ORGANIZATION_BLOCK MAIN:OB1
TITLE=中文详细注释版
// 文件说明：本文件只完善中文注释，不改变 PLC 指令、地址和执行顺序。
// 编码说明：本文件采用 GBK/ANSI 编码，供现场 PLC 编辑环境直接打开。
//
// ======================== 本项目工序与地址总表 ========================
// 说明：“程序网络 N”是 AWL Network 编号，不等于设备主屏上的工序序号。
// 主工序顺序（与上位机主屏一致）：
//   等待启动(M0.0=0) -> 初始位垂直复位(M10.0) -> 初始位确认(M10.1)
//   -> 检测区1定位(M10.2) -> 热源位夹具下压(M10.3) -> 30秒稳定 -> 30秒噪声采集(M25.2)
//   -> 热源干扰测试(M10.4)
//   -> 热源后夹具上升(M10.5) -> 检测区2定位(M10.6) -> 爆闪位夹具下压(M10.7)
//   -> 五次爆闪测试(M11.0) -> 电磁干扰(M11.2) -> 回初始位确认(M11.4)
//   -> 流程完成(M0.1)。
//
// 输入 I（现场反馈/命令）：
//   I0.0 初始位置传感器；I0.2 检测区1位置传感器；I0.1 检测区2位置传感器。
//   I0.4 垂直下限反馈；I0.3 垂直上限反馈（本版主链以定时到位为主，地址保留作项目对照）。
//   I1.0 安全/急停输入：1=安全链满足，0=急停或安全链断开。
//   I1.3 自动启动输入：闭合上升沿触发一次完整检测工序。
//
// 物理输出继电器 Q（与主屏“输出继电器 Q”一致）：
//   Q0.0 预留/本程序无独立驱动，仅在总复位时清零。
//   Q0.1 模拟人温度/热源；Q0.2、Q0.3 预留/本程序无独立驱动。
//   Q0.4 上下电机总电源；Q0.5 左右电机运行；Q0.6 左右电机停止。
//   Q0.7 电磁干扰继电器，实际链路为 M11.2 AND M31.7 -> Q0.7。
//   Q1.0 气缸/挥手测试；Q1.1 垂直方向（1=上，0=下）。
//   Q1.2 爆闪灯1；Q1.3 爆闪灯2。
//
// 主状态与启动/停止辅助继电器 M：
//   M0.0 自动运行；M0.1 流程完成；M0.2 流程报警；M0.3 安全链满足。
//   M1.0 停止/中止锁存；M1.2 启动条件确认后的单扫描启动脉冲。
//   M1.5 启动请求上一扫描状态；M1.6 启动请求上升沿；M1.7 手动使能启动通道。
//   M2.0 停止请求；M2.1 总复位/初始化请求；M2.2 安全限位；
//   M2.3 启动请求；M2.4 手动使能。M20.0 为安全链断开故障镜像。
//
// 主工序步进继电器（同一时刻通常只保持当前工序位）：
//   M10.0 初始位垂直复位；M10.1 初始位确认；M10.2 检测区1定位。
//   M10.3 热源位夹具下压；M10.4 热源干扰测试；M10.5 热源后夹具上升。
//   M10.6 检测区2定位；M10.7 爆闪位夹具下压；M11.0 五次爆闪测试。
//   M11.1 外部/备用的电磁工序启动脉冲；M11.2 电磁干扰工序控制位；
//   M11.3 回零完成后的流程结束脉冲；M11.4 电磁干扰后回初始位标志。
//
// 工序完成条件与动作子步：
//   M12.0 初始垂直复位延时完成；M12.1 初始位置确认；M12.2 检测区1到位。
//   M12.3 热源位夹具下压延时完成；M12.5 热源后夹具上升延时完成；
//   M12.6 检测区2到位；M12.7 爆闪位夹具下压延时完成。
//   M13.0~M13.4 热源干扰时的气缸/挥手脉冲子步（开、关交替）。
//   M13.5~M15.7 五次爆闪时序子步；奇数发光段驱动 Q1.2、Q1.3，间隔段熄灯。
//   M14.0 初始复位后的重叠移动等待；M14.1 初始位至检测区1的启动等待；
//   M14.2 检测区1到位后的下压启动等待；M14.3 上升后的水平移动等待（预留链）；
//   M14.4 检测区2到位后的下压启动等待。
//   M15.0 热源位下压后的稳定等待标志；M15.1 爆闪位下压后的稳定等待标志；
//   M15.2 热源测试后“垂直上升+水平移向检测区2”的重叠动作标志；
//   M15.3 热源夹具上升完成、等待进入检测区2下压的衔接标志。
//
// 上位机/通讯状态与事件留痕位：
//   M21.0 初始位阶段；M21.1 检测区1/热源阶段；M21.2 检测区2/爆闪阶段；
//   M21.3 电磁干扰阶段；M21.4 初始位置已确认；M21.5 热源后夹具已上升；
//   M21.6 五次爆闪已完成；M21.7 电磁干扰已完成。
//   M22.0 初始垂直复位完成；M22.1、M22.2 初始位置确认留痕；
//   M22.3 检测区1到位；M22.4 热源位下压完成；M22.5 热源干扰完成；
//   M22.6 爆闪位下压完成；M22.7 运动到位/衔接留痕（由上升或检测区2到位置位）。
//   M23.0 五次爆闪完成；M23.1 电磁干扰开始；M23.2 电磁干扰完成；
//   M23.3 电磁干扰完成后开始回初始位。
//
// 自动/手动动作命令、沿检测及安全合成：
//   M29.0 自动左右运行；M29.1 自动垂直下行；M29.2 自动垂直上行；
//   M29.3 自动气缸/挥手；M29.4 自动爆闪命令（当前五次爆闪另由时序子步直接合成）。
//   M30.0~M30.6 手动/调试动作命令；M30.7 手动总停止/全部输出清零。
//   M28.0~M28.4 保存 M29.0~M29.4 的上一扫描状态；
//   M26.0~M26.4 为相应自动动作的上升沿，M27.0~M27.4 为下降沿；
//   M26.5 为任一自动动作上升沿，M27.5 为垂直上/下动作结束的互锁辅助位。
//   M31.0 热源输出合成；M31.1 垂直电源合成；M31.2 垂直向上方向合成；
//   M31.3 水平运行合成；M31.4 水平停止合成；M31.5 爆闪灯1合成；
//   M31.6 爆闪灯2合成；M31.7 总输出安全使能（安全链满足且无手动总停止）。
//   M25.0 安全限位上升沿单扫描脉冲；M25.1 正常水平停止请求；
//   M25.2 为信号稳定后的30秒噪声采集窗口，由 T63 稳定到时后直接驱动。
//
// 状态字：VW600=上位机工序阶段码；VW602=上位机工序子步码。
//
// ======================== 定时器实际时间参数表 ========================
// 计时规则：本程序全部使用 TON T37~T63；按 S7-200 SMART 定时器规则，
//           T37~T63 的时间基准均为 100 ms，实际延迟 = PT预置值 x 0.1秒。
//           下表按本文件当前 PT 值换算；修改 PT 后必须同步更新此表及网络注释。
//
// 初始位、定位及夹具动作：
//   T44  初始位垂直复位动作延时       PT=+20   -> 2.0秒
//   T45  热源位夹具下压动作延时       PT=+100  -> 10.0秒
//   T46  热源测试后夹具上升动作延时   PT=+100  -> 10.0秒
//   T47  爆闪位夹具下压动作延时       PT=+100  -> 10.0秒
//
// 工序切换及机械稳定等待：
//   T48  初始复位后的重叠移动等待     PT=+80   -> 8.0秒
//   T49  初始位至检测区1启动等待      PT=+10   -> 1.0秒
//   T50  检测区1到位后的下压启动等待  PT=+10   -> 1.0秒
//   T51  信号稳定后噪声采集窗口   PT=+300  -> 30.0秒
//   T52  检测区2到位后的下压切换等待  PT=+10   -> 1.0秒
//   T62  垂直上升与水平移动重叠许可   PT=+20   -> 2.0秒
//   T63  热源位夹具下压后的稳定等待 PT=+300  -> 30.0秒
//   T38  爆闪位夹具下压后的稳定等待 PT=+100  -> 10.0秒
//
// 热源干扰/气缸挥手节拍：
//   T37、T40、T41、T42、T43 每段 PT=+10 -> 每段1.0秒；
//   共5段、总时序约5.0秒，形成3次动作段与2次间隔段。
//
// 五次爆闪节拍：
//   T53~T61 共9段，每段 PT=+10 -> 每段1.0秒；
//   总时序约9.0秒，形成5次亮灯段与4次灭灯间隔段。
//
// 电磁干扰：
//   T39  电磁干扰继电器 Q0.7 保持时间 PT=+100 -> 10.0秒。
// ======================================================================
// ======================================================================
BEGIN
// ----------------------------------------------------------------------
// 安全链、报警及复位总控
// ----------------------------------------------------------------------
Network 1
// 程序网络 1：把安全/急停输入 I1.0 映射为“安全链满足”M0.3。
// 输入状态初始化。
// 装载 I1.0 的状态，作为当前逻辑判断起点。
LD     I1.0
// 将当前逻辑结果写入 M0.3。
=      M0.3
Network 2
// 程序网络 2：安全链断开或收到停止请求时，生成停止/中止锁存 M1.0。
// 装载 I1.0 的反状态，作为当前逻辑判断起点。
LDN    I1.0
// 与 M2.0 进行并联“或”条件判断。
O      M2.0
// 将当前逻辑结果写入 M1.0。
=      M1.0
Network 3
// 程序网络 3：将安全链断开状态镜像到故障辅助位 M20.0。
// 装载 I1.0 的反状态，作为当前逻辑判断起点。
LDN    I1.0
// 将当前逻辑结果写入 M20.0。
=      M20.0
Network 4
// 程序网络 4：安全链断开时置流程报警 M0.2。
// 装载 M20.0 的状态，作为当前逻辑判断起点。
LD     M20.0
// 将当前逻辑结果写入 M0.2。
=      M0.2
Network 5
// 程序网络 5：执行流程条件判断与状态控制。
// 装载 M2.1 的状态，作为当前逻辑判断起点。
LD     M2.1
// 条件成立时复位 M0.0，连续复位 3 位。
R      M0.0, 3
Network 6
// 程序网络 6：满足条件时执行批量复位/停止处理。
// 装载 M2.1 的状态，作为当前逻辑判断起点。
LD     M2.1
// 条件成立时复位 M10.0，连续复位 12 位。
R      M10.0, 12
// 条件成立时复位 M11.4，连续复位 1 位。
R      M11.4, 1
// 条件成立时复位 M13.0，连续复位 8 位。
R      M13.0, 8
// 条件成立时复位 M14.0，连续复位 8 位。
R      M14.0, 8
// 条件成立时复位 M15.0，连续复位 4 位。
R      M15.0, 4
// 条件成立时复位 M15.4，连续复位 4 位。
R      M15.4, 4
Network 7
// 程序网络 7：执行流程条件判断与状态控制。
// 装载 M2.1 的状态，作为当前逻辑判断起点。
LD     M2.1
// 条件成立时复位 M12.0，连续复位 10 位。
R      M12.0, 10
Network 8
// 程序网络 8：满足条件时执行批量复位/停止处理。
// 装载 M2.1 的状态，作为当前逻辑判断起点。
LD     M2.1
// 条件成立时复位 M21.0，连续复位 8 位。
R      M21.0, 8
// 条件成立时复位 M29.0，连续复位 8 位。
R      M29.0, 8
// 条件成立时复位 M30.0，连续复位 8 位。
R      M30.0, 8
// 条件成立时复位 Q0.0，连续复位 8 位。
R      Q0.0, 8
// 条件成立时复位 Q1.0，连续复位 4 位。
R      Q1.0, 4
Network 9
// 程序网络 9：执行流程条件判断与状态控制。
// 装载 M2.1 的状态，作为当前逻辑判断起点。
LD     M2.1
// 条件成立时复位 M22.0，连续复位 12 位。
R      M22.0, 12
Network 10
// 程序网络 10：执行流程条件判断与状态控制。
// 装载 M2.1 的状态，作为当前逻辑判断起点。
LD     M2.1
// 条件成立时复位 M20.0，连续复位 1 位。
R      M20.0, 1
Network 11
// 程序网络 11：更新流程状态字或显示/通讯状态值。
// 装载 M2.1 的状态，作为当前逻辑判断起点。
LD     M2.1
// 条件成立时将字数据 +0 写入 VW600。
MOVW   +0, VW600
Network 12
// 程序网络 12：更新流程状态字或显示/通讯状态值。
// 装载 M2.1 的状态，作为当前逻辑判断起点。
LD     M2.1
// 条件成立时将字数据 +0 写入 VW602。
MOVW   +0, VW602
Network 13
// 程序网络 13：执行流程条件判断与状态控制。
// 装载 M1.0 的状态，作为当前逻辑判断起点。
LD     M1.0
// 条件成立时复位 M0.0，连续复位 1 位。
R      M0.0, 1
Network 14
// 程序网络 14：满足条件时执行批量复位/停止处理。
// 装载 M1.0 的状态，作为当前逻辑判断起点。
LD     M1.0
// 条件成立时复位 M10.0，连续复位 12 位。
R      M10.0, 12
// 条件成立时复位 M11.4，连续复位 1 位。
R      M11.4, 1
// 条件成立时复位 M13.0，连续复位 8 位。
R      M13.0, 8
// 条件成立时复位 M14.0，连续复位 8 位。
R      M14.0, 8
// 条件成立时复位 M15.0，连续复位 4 位。
R      M15.0, 4
// 条件成立时复位 M15.4，连续复位 4 位。
R      M15.4, 4
Network 15
// 程序网络 15：执行流程条件判断与状态控制。
// 装载 M1.0 的状态，作为当前逻辑判断起点。
LD     M1.0
// 条件成立时复位 M12.0，连续复位 10 位。
R      M12.0, 10
Network 16
// 程序网络 16：满足条件时执行批量复位/停止处理。
// 装载 M1.0 的状态，作为当前逻辑判断起点。
LD     M1.0
// 条件成立时复位 M21.0，连续复位 8 位。
R      M21.0, 8
// 条件成立时复位 M22.0，连续复位 12 位。
R      M22.0, 12
// 条件成立时复位 M29.0，连续复位 8 位。
R      M29.0, 8
// 条件成立时复位 M30.0，连续复位 8 位。
R      M30.0, 8
// 条件成立时复位 Q0.0，连续复位 8 位。
R      Q0.0, 8
// 条件成立时复位 Q1.0，连续复位 4 位。
R      Q1.0, 4
Network 17
// 程序网络 17：更新流程状态字或显示/通讯状态值。
// 装载 M1.0 的状态，作为当前逻辑判断起点。
LD     M1.0
// 条件成立时将字数据 +0 写入 VW600。
MOVW   +0, VW600
Network 18
// 程序网络 18：更新流程状态字或显示/通讯状态值。
// 装载 M1.0 的状态，作为当前逻辑判断起点。
LD     M1.0
// 条件成立时将字数据 +0 写入 VW602。
MOVW   +0, VW602
// ----------------------------------------------------------------------
// 启动请求沿检测与自动流程起动
// ----------------------------------------------------------------------
Network 19
// 程序网络 19：组合条件并生成状态或输出结果。
// 装载 M2.3 的状态，作为当前逻辑判断起点。
LD     M2.3
// 与 M1.5 的反状态进行串联条件判断。
AN     M1.5
// 将当前逻辑结果写入 M1.6。
=      M1.6
Network 20
// 程序网络 20：组合条件并生成状态或输出结果。
// 装载 M2.3 的状态，作为当前逻辑判断起点。
LD     M2.3
// 将当前逻辑结果写入 M1.5。
=      M1.5
Network 21
// 程序网络 21：组合条件并生成状态或输出结果。
// 装载 M1.6 的状态，作为当前逻辑判断起点。
LD     M1.6
// 与 M2.4 进行串联条件判断。
A      M2.4
// 与 M0.3 进行串联条件判断。
A      M0.3
// 将当前逻辑结果写入 M1.7。
=      M1.7
Network 22
// 程序网络 22：合成自动/手动启动条件，输出一次启动确认脉冲 M1.2。
// I1.3 上升沿通过正常安全联锁后启动自动流程。
// 装载 M1.6 的状态，作为当前逻辑判断起点。
LD     M1.6
// 与 M0.3 进行串联条件判断。
A      M0.3
// 与 M0.2 的反状态进行串联条件判断。
AN     M0.2
// 与 M0.0 的反状态进行串联条件判断。
AN     M0.0
// 与 M1.7 进行并联“或”条件判断。
O      M1.7
// 装载 I1.3 的状态，作为当前逻辑判断起点。
LD     I1.3
// 检测当前逻辑结果的上升沿，仅在上升沿扫描周期成立。
EU
// 与 M0.3 进行串联条件判断。
A      M0.3
// 与 M0.2 的反状态进行串联条件判断。
AN     M0.2
// 与 M0.0 的反状态进行串联条件判断。
AN     M0.0
// 将当前逻辑块与前一逻辑块进行“或”运算。
OLD
// 将当前逻辑结果写入 M1.2。
=      M1.2
Network 23
// 程序网络 23：执行流程条件判断与状态控制。
// 装载 M1.2 的状态，作为当前逻辑判断起点。
LD     M1.2
// 条件成立时置位 M0.0，连续置位 1 位。
S      M0.0, 1
Network 24
// 程序网络 24：执行流程条件判断与状态控制。
// 装载 M1.2 的状态，作为当前逻辑判断起点。
LD     M1.2
// 条件成立时复位 M0.1，连续复位 1 位。
R      M0.1, 1
Network 25
// 程序网络 25：满足条件时执行批量复位/停止处理。
// 装载 M1.2 的状态，作为当前逻辑判断起点。
LD     M1.2
// 条件成立时复位 M10.0，连续复位 12 位。
R      M10.0, 12
// 条件成立时复位 M11.4，连续复位 1 位。
R      M11.4, 1
// 条件成立时复位 M13.0，连续复位 8 位。
R      M13.0, 8
// 条件成立时复位 M14.0，连续复位 8 位。
R      M14.0, 8
// 条件成立时复位 M15.0，连续复位 4 位。
R      M15.0, 4
// 条件成立时复位 M15.4，连续复位 4 位。
R      M15.4, 4
Network 26
// 程序网络 26：执行流程条件判断与状态控制。
// 装载 M1.2 的状态，作为当前逻辑判断起点。
LD     M1.2
// 条件成立时复位 M2.0，连续复位 1 位。
R      M2.0, 1
Network 27
// 程序网络 27：满足条件时执行批量复位/停止处理。
// 装载 M1.2 的状态，作为当前逻辑判断起点。
LD     M1.2
// 条件成立时复位 M21.0，连续复位 8 位。
R      M21.0, 8
// 条件成立时复位 M29.0，连续复位 8 位。
R      M29.0, 8
// 条件成立时复位 M30.0，连续复位 8 位。
R      M30.0, 8
// 条件成立时复位 Q0.0，连续复位 8 位。
R      Q0.0, 8
// 条件成立时复位 Q1.0，连续复位 4 位。
R      Q1.0, 4
Network 28
// 程序网络 28：执行流程条件判断与状态控制。
// 装载 M1.2 的状态，作为当前逻辑判断起点。
LD     M1.2
// 条件成立时复位 M22.0，连续复位 12 位。
R      M22.0, 12
Network 29
// 程序网络 29：启动后进入“初始位垂直复位”M10.0，并发出自动上行 M29.2。
// 装载 M1.2 的状态，作为当前逻辑判断起点。
LD     M1.2
// 条件成立时置位 M10.0，连续置位 1 位。
S      M10.0, 1
// 条件成立时置位 M29.2，连续置位 1 位。
S      M29.2, 1
Network 30
// 程序网络 30：更新流程状态字或显示/通讯状态值。
// 装载 M1.2 的状态，作为当前逻辑判断起点。
LD     M1.2
// 条件成立时将字数据 +1 写入 VW600。
MOVW   +1, VW600
Network 31
// 程序网络 31：更新流程状态字或显示/通讯状态值。
// 装载 M1.2 的状态，作为当前逻辑判断起点。
LD     M1.2
// 条件成立时将字数据 +1 写入 VW602。
MOVW   +1, VW602
// ----------------------------------------------------------------------
// 主工序完成条件、延时及到位判定
// ----------------------------------------------------------------------
Network 32
// 程序网络 32：执行流程条件判断与状态控制。
// 装载 M10.1 的状态，作为当前逻辑判断起点。
LD     M10.1
// 与 M10.2 进行并联“或”条件判断。
O      M10.2
// 与 M10.6 进行并联“或”条件判断。
O      M10.6
// 条件成立时复位 Q0.6，连续复位 1 位。
R      Q0.6, 1
// 条件成立时置位 M29.0，连续置位 1 位。
S      M29.0, 1
Network 33
// 程序网络 33：初始位垂直复位动作计时 T44。
// 垂直机构初始化：先执行上行定时，再与水平回零流程进行重叠动作。
// 装载 M10.0 的状态，作为当前逻辑判断起点。
LD     M10.0
// T44（初始位垂直复位动作延时）：PT=+20，时间基准=100 ms，实际延迟=2.0秒。
TON    T44, +20
Network 34
// 程序网络 34：T44 到时，生成初始垂直复位完成 M12.0。
// 装载 T44 的状态，作为当前逻辑判断起点。
LD     T44
// 将当前逻辑结果写入 M12.0。
=      M12.0
Network 35
// 程序网络 35：M10.1 期间检测 I0.0，确认设备已在初始水平位置。
// 装载 M10.1 的状态，作为当前逻辑判断起点。
LD     M10.1
// 与 I0.0 进行串联条件判断。
A      I0.0
// 将当前逻辑结果写入 M12.1。
=      M12.1
Network 36
// 程序网络 36：M10.2 期间检测 I0.2，确认已到检测区1。
// 装载 M10.2 的状态，作为当前逻辑判断起点。
LD     M10.2
// 与 I0.2 进行串联条件判断。
A      I0.2
// 将当前逻辑结果写入 M12.2。
=      M12.2
Network 37
// 程序网络 37：热源位夹具下压动作计时 T45。
// 装载 M10.3 的状态，作为当前逻辑判断起点。
LD     M10.3
// T45（热源位夹具下压动作延时）：PT=+100，时间基准=100 ms，实际延迟=10.0秒。
TON    T45, +100
Network 38
// 程序网络 38：T45 到时，生成热源位夹具下压完成 M12.3。
// 装载 T45 的状态，作为当前逻辑判断起点。
LD     T45
// 将当前逻辑结果写入 M12.3。
=      M12.3
Network 39
// 程序网络 39：热源测试后夹具上升动作计时 T46。
// 装载 M10.5 的状态，作为当前逻辑判断起点。
LD     M10.5
// T46（热源测试后夹具上升动作延时）：PT=+100，时间基准=100 ms，实际延迟=10.0秒。
TON    T46, +100
Network 40
// 程序网络 40：T46 到时，生成热源后夹具上升完成 M12.5。
// 装载 T46 的状态，作为当前逻辑判断起点。
LD     T46
// 将当前逻辑结果写入 M12.5。
=      M12.5
Network 41
// 程序网络 41：M10.6 期间检测 I0.1，确认已到检测区2。
// 装载 M10.6 的状态，作为当前逻辑判断起点。
LD     M10.6
// 与 I0.1 进行串联条件判断。
A      I0.1
// 将当前逻辑结果写入 M12.6。
=      M12.6
Network 42
// 程序网络 42：爆闪位夹具下压动作计时 T47。
// 装载 M10.7 的状态，作为当前逻辑判断起点。
LD     M10.7
// T47（爆闪位夹具下压动作延时）：PT=+100，时间基准=100 ms，实际延迟=10.0秒。
TON    T47, +100
Network 43
// 程序网络 43：T47 到时，生成爆闪位夹具下压完成 M12.7。
// 装载 T47 的状态，作为当前逻辑判断起点。
LD     T47
// 将当前逻辑结果写入 M12.7。
=      M12.7
Network 44
// 程序网络 44：定时与条件控制，涉及 T48。
// 装载 M14.0 的状态，作为当前逻辑判断起点。
LD     M14.0
// T48（初始复位后的重叠移动等待）：PT=+80，时间基准=100 ms，实际延迟=8.0秒。
TON    T48, +80
Network 45
// 程序网络 45：定时与条件控制，涉及 T49。
// 装载 M14.1 的状态，作为当前逻辑判断起点。
LD     M14.1
// T49（初始位至检测区1启动等待）：PT=+10，时间基准=100 ms，实际延迟=1.0秒。
TON    T49, +10
Network 46
// 程序网络 46：定时与条件控制，涉及 T50。
// 装载 M14.2 的状态，作为当前逻辑判断起点。
LD     M14.2
// T50（检测区1到位后的下压启动等待）：PT=+10，时间基准=100 ms，实际延迟=1.0秒。
TON    T50, +10
Network 47
// 程序网络 47：M25.2 置位后开始独立的30秒噪声采集定时。
LD     M25.2
// T51（噪声采集窗口）：PT=+300，时间基准=100 ms，实际延迟=30.0秒。
TON    T51, +300
Network 48
// 程序网络 48：定时与条件控制，涉及 T52、T62、T63、T38。
// 全局垂直上行重叠许可：T62 到时后允许水平与垂直动作重叠。
// 热源位夹紧下压完成后先稳定30秒，再置位 M25.2 开始30秒噪声采集。
// 装载 M14.4 的状态，作为当前逻辑判断起点。
LD     M14.4
// 与 M15.3 进行串联条件判断。
A      M15.3
// T52（检测区2到位后的下压切换等待）：PT=+10，时间基准=100 ms，实际延迟=1.0秒。
TON    T52, +10
// 装载 M29.2 的状态，作为当前逻辑判断起点。
LD     M29.2
// T62（垂直上升与水平移动重叠许可）：PT=+20，时间基准=100 ms，实际延迟=2.0秒。
TON    T62, +20
// 装载 M15.0 的状态，作为当前逻辑判断起点。
LD     M15.0
// T63（热源位稳定等待）：PT=+300，时间基准=100 ms，实际延迟=30.0秒。
TON    T63, +300
// 稳定完成且仍处于热源位等待状态时，发布噪声采集窗口。
LD     T63
A      M15.0
=      M25.2
// 爆闪位使用独立的10秒稳定定时，不与热源噪声窗口共用。
LD     M15.1
TON    T38, +100
// ----------------------------------------------------------------------
// 主步进链：初始位 -> 检测区1 -> 热源测试 -> 检测区2
// ----------------------------------------------------------------------
Network 49
// 程序网络 49：执行流程条件判断与状态控制。
// 装载 M12.0 的状态，作为当前逻辑判断起点。
LD     M12.0
// 条件成立时复位 M10.0，连续复位 1 位。
R      M10.0, 1
Network 50
// 程序网络 50：满足条件时置位多个流程状态。
// 装载 M12.0 的状态，作为当前逻辑判断起点。
LD     M12.0
// 条件成立时置位 M14.0，连续置位 1 位。
S      M14.0, 1
// 条件成立时置位 M10.1，连续置位 1 位。
S      M10.1, 1
// 条件成立时置位 M29.0，连续置位 1 位。
S      M29.0, 1
Network 51
// 程序网络 51：满足条件时执行批量复位/停止处理。
// 装载 T48 的状态，作为当前逻辑判断起点。
LD     T48
// 条件成立时复位 M14.0，连续复位 1 位。
R      M14.0, 1
// 条件成立时复位 M29.2，连续复位 1 位。
R      M29.2, 1
Network 52
// 程序网络 52：执行流程条件判断与状态控制。
// 装载 T48 的状态，作为当前逻辑判断起点。
LD     T48
// 条件成立时复位 Q0.6，连续复位 1 位。
R      Q0.6, 1
Network 53
// 程序网络 53：执行流程条件判断与状态控制。
// 装载 M12.0 的状态，作为当前逻辑判断起点。
LD     M12.0
// 条件成立时置位 M22.0，连续置位 1 位。
S      M22.0, 1
Network 54
// 程序网络 54：更新流程状态字或显示/通讯状态值。
// 装载 M12.0 的状态，作为当前逻辑判断起点。
LD     M12.0
// 条件成立时将字数据 +1 写入 VW602。
MOVW   +1, VW602
Network 55
// 程序网络 55：满足条件时执行批量复位/停止处理。
// 装载 M12.1 的状态，作为当前逻辑判断起点。
LD     M12.1
// 条件成立时复位 M10.1，连续复位 1 位。
R      M10.1, 1
// 条件成立时复位 M29.0，连续复位 1 位。
R      M29.0, 1
Network 56
// 程序网络 56：执行流程条件判断与状态控制。
// 装载 M12.1 的状态，作为当前逻辑判断起点。
LD     M12.1
// 条件成立时置位 M14.1，连续置位 1 位。
S      M14.1, 1
Network 57
// 程序网络 57：执行流程条件判断与状态控制。
// 装载 T49 的状态，作为当前逻辑判断起点。
LD     T49
// 条件成立时复位 M14.1，连续复位 1 位。
R      M14.1, 1
Network 58
// 程序网络 58：满足条件时置位多个流程状态。
// 装载 T49 的状态，作为当前逻辑判断起点。
LD     T49
// 与 M11.4 的反状态进行串联条件判断。
AN     M11.4
// 条件成立时复位 Q0.6，连续复位 1 位。
R      Q0.6, 1
// 条件成立时置位 M10.2，连续置位 1 位。
S      M10.2, 1
// 条件成立时置位 M29.0，连续置位 1 位。
S      M29.0, 1
Network 59
// 程序网络 59：满足条件时置位多个流程状态。
// 装载 T49 的状态，作为当前逻辑判断起点。
LD     T49
// 与 M11.4 进行串联条件判断。
A      M11.4
// 条件成立时置位 M11.3，连续置位 1 位。
S      M11.3, 1
// 条件成立时置位 M2.0，连续置位 1 位。
S      M2.0, 1
// 条件成立时复位 M11.4，连续复位 1 位。
R      M11.4, 1
Network 60
// 程序网络 60：执行流程条件判断与状态控制。
// 装载 M12.1 的状态，作为当前逻辑判断起点。
LD     M12.1
// 条件成立时置位 M22.1，连续置位 1 位。
S      M22.1, 1
Network 61
// 程序网络 61：执行流程条件判断与状态控制。
// 装载 M12.1 的状态，作为当前逻辑判断起点。
LD     M12.1
// 条件成立时置位 M22.2，连续置位 1 位。
S      M22.2, 1
Network 62
// 程序网络 62：执行流程条件判断与状态控制。
// 装载 M12.1 的状态，作为当前逻辑判断起点。
LD     M12.1
// 条件成立时置位 M21.4，连续置位 1 位。
S      M21.4, 1
Network 63
// 程序网络 63：更新流程状态字或显示/通讯状态值。
// 装载 M12.1 的状态，作为当前逻辑判断起点。
LD     M12.1
// 条件成立时将字数据 +2 写入 VW600。
MOVW   +2, VW600
Network 64
// 程序网络 64：更新流程状态字或显示/通讯状态值。
// 装载 M12.1 的状态，作为当前逻辑判断起点。
LD     M12.1
// 条件成立时将字数据 +2 写入 VW602。
MOVW   +2, VW602
Network 65
// 程序网络 65：满足条件时执行批量复位/停止处理。
// 装载 M12.2 的状态，作为当前逻辑判断起点。
LD     M12.2
// 条件成立时复位 M10.2，连续复位 1 位。
R      M10.2, 1
// 条件成立时复位 M29.0，连续复位 1 位。
R      M29.0, 1
// 条件成立时置位 Q0.6，连续置位 1 位。
S      Q0.6, 1
Network 66
// 程序网络 66：执行流程条件判断与状态控制。
// 装载 M12.2 的状态，作为当前逻辑判断起点。
LD     M12.2
// 条件成立时置位 M14.2，连续置位 1 位。
S      M14.2, 1
Network 67
// 程序网络 67：执行流程条件判断与状态控制。
// 装载 T50 的状态，作为当前逻辑判断起点。
LD     T50
// 条件成立时复位 M14.2，连续复位 1 位。
R      M14.2, 1
Network 68
// 程序网络 68：满足条件时置位多个流程状态。
// 装载 T50 的状态，作为当前逻辑判断起点。
LD     T50
// 条件成立时置位 M10.3，连续置位 1 位。
S      M10.3, 1
// 条件成立时置位 M29.1，连续置位 1 位。
S      M29.1, 1
Network 69
// 程序网络 69：执行流程条件判断与状态控制。
// 装载 M12.2 的状态，作为当前逻辑判断起点。
LD     M12.2
// 条件成立时置位 M22.3，连续置位 1 位。
S      M22.3, 1
Network 70
// 程序网络 70：更新流程状态字或显示/通讯状态值。
// 装载 M12.2 的状态，作为当前逻辑判断起点。
LD     M12.2
// 条件成立时将字数据 +2 写入 VW602。
MOVW   +2, VW602
Network 71
// 程序网络 71：执行流程条件判断与状态控制。
// 装载 M12.3 的状态，作为当前逻辑判断起点。
LD     M12.3
// 条件成立时复位 M10.3，连续复位 1 位。
R      M10.3, 1
Network 72
// 程序网络 72：执行流程条件判断与状态控制。
// 装载 M12.3 的状态，作为当前逻辑判断起点。
LD     M12.3
R      M29.1, 1
// 条件成立时置位 M15.0，连续置位 1 位。
S      M15.0, 1
Network 73
// 程序网络 73：执行流程条件判断与状态控制。
// 装载 M12.3 的状态，作为当前逻辑判断起点。
LD     M12.3
// 条件成立时置位 M22.4，连续置位 1 位。
S      M22.4, 1
// ----------------------------------------------------------------------
// 热源干扰测试：夹具稳定后执行气缸/挥手节拍
// ----------------------------------------------------------------------
Network 74
// 程序网络 74：夹具稳定等待结束后进入热源干扰测试，并启动首个气缸/挥手脉冲。
// 等待 T51 完成整30秒噪声采集后，再启动加热测试。
// 装载 M12.3 的状态，作为当前逻辑判断起点。
LD     M12.3
// 条件成立时将字数据 +3 写入 VW602。
MOVW   +3, VW602
// 装载 T51 的状态，作为当前逻辑判断起点。
LD     T51
// 与 M15.0 进行串联条件判断。
A      M15.0
// 条件成立时复位 M15.0，连续复位 1 位。
R      M15.0, 1
// 条件成立时置位 M10.4，连续置位 1 位。
S      M10.4, 1
// 条件成立时置位 M13.0，连续置位 1 位。
S      M13.0, 1
// 条件成立时置位 M29.3，连续置位 1 位。
S      M29.3, 1
Network 75
// 程序网络 75：定时与条件控制，涉及 T37。
// 装载 M13.0 的状态，作为当前逻辑判断起点。
LD     M13.0
// T37（热源干扰第1段气缸/挥手节拍）：PT=+10，时间基准=100 ms，实际延迟=1.0秒。
TON    T37, +10
Network 76
// 程序网络 76：满足条件时执行批量复位/停止处理。
// 装载 T37 的状态，作为当前逻辑判断起点。
LD     T37
// 条件成立时复位 M13.0，连续复位 1 位。
R      M13.0, 1
// 条件成立时复位 M29.3，连续复位 1 位。
R      M29.3, 1
Network 77
// 程序网络 77：执行流程条件判断与状态控制。
// 装载 T37 的状态，作为当前逻辑判断起点。
LD     T37
// 条件成立时置位 M13.1，连续置位 1 位。
S      M13.1, 1
Network 78
// 程序网络 78：定时与条件控制，涉及 T40。
// 装载 M13.1 的状态，作为当前逻辑判断起点。
LD     M13.1
// T40（热源干扰第2段气缸/挥手节拍）：PT=+10，时间基准=100 ms，实际延迟=1.0秒。
TON    T40, +10
Network 79
// 程序网络 79：执行流程条件判断与状态控制。
// 装载 T40 的状态，作为当前逻辑判断起点。
LD     T40
// 条件成立时复位 M13.1，连续复位 1 位。
R      M13.1, 1
Network 80
// 程序网络 80：满足条件时置位多个流程状态。
// 装载 T40 的状态，作为当前逻辑判断起点。
LD     T40
// 条件成立时置位 M13.2，连续置位 1 位。
S      M13.2, 1
// 条件成立时置位 M29.3，连续置位 1 位。
S      M29.3, 1
Network 81
// 程序网络 81：定时与条件控制，涉及 T41。
// 装载 M13.2 的状态，作为当前逻辑判断起点。
LD     M13.2
// T41（热源干扰第3段气缸/挥手节拍）：PT=+10，时间基准=100 ms，实际延迟=1.0秒。
TON    T41, +10
Network 82
// 程序网络 82：满足条件时执行批量复位/停止处理。
// 装载 T41 的状态，作为当前逻辑判断起点。
LD     T41
// 条件成立时复位 M13.2，连续复位 1 位。
R      M13.2, 1
// 条件成立时复位 M29.3，连续复位 1 位。
R      M29.3, 1
Network 83
// 程序网络 83：执行流程条件判断与状态控制。
// 装载 T41 的状态，作为当前逻辑判断起点。
LD     T41
// 条件成立时置位 M13.3，连续置位 1 位。
S      M13.3, 1
Network 84
// 程序网络 84：定时与条件控制，涉及 T42。
// 装载 M13.3 的状态，作为当前逻辑判断起点。
LD     M13.3
// T42（热源干扰第4段气缸/挥手节拍）：PT=+10，时间基准=100 ms，实际延迟=1.0秒。
TON    T42, +10
Network 85
// 程序网络 85：执行流程条件判断与状态控制。
// 装载 T42 的状态，作为当前逻辑判断起点。
LD     T42
// 条件成立时复位 M13.3，连续复位 1 位。
R      M13.3, 1
Network 86
// 程序网络 86：满足条件时置位多个流程状态。
// 装载 T42 的状态，作为当前逻辑判断起点。
LD     T42
// 条件成立时置位 M13.4，连续置位 1 位。
S      M13.4, 1
// 条件成立时置位 M29.3，连续置位 1 位。
S      M29.3, 1
Network 87
// 程序网络 87：定时与条件控制，涉及 T43。
// 装载 M13.4 的状态，作为当前逻辑判断起点。
LD     M13.4
// T43（热源干扰第5段气缸/挥手节拍）：PT=+10，时间基准=100 ms，实际延迟=1.0秒。
TON    T43, +10
Network 88
// 程序网络 88：满足条件时执行批量复位/停止处理。
// 装载 T43 的状态，作为当前逻辑判断起点。
LD     T43
// 条件成立时复位 M13.4，连续复位 1 位。
R      M13.4, 1
// 条件成立时复位 M10.4，连续复位 1 位。
R      M10.4, 1
// 条件成立时复位 M29.3，连续复位 1 位。
R      M29.3, 1
Network 89
// 程序网络 89：热源挥手节拍结束，进入“热源后夹具上升”并发出自动上行命令。
// 装载 T43 的状态，作为当前逻辑判断起点。
LD     T43
// 条件成立时复位 M15.2，连续复位 2 位。
R      M15.2, 2
// 条件成立时置位 M10.5，连续置位 1 位。
S      M10.5, 1
// 条件成立时置位 M29.2，连续置位 1 位。
S      M29.2, 1
Network 90
// 程序网络 90：执行流程条件判断与状态控制。
// 装载 T43 的状态，作为当前逻辑判断起点。
LD     T43
// 条件成立时置位 M22.5，连续置位 1 位。
S      M22.5, 1
Network 91
// 程序网络 91：上升许可延时满足后，重叠启动向检测区2的水平移动。
// 垂直上行延时满足后，仅触发一次水平移动，同时保持垂直上行动作。
// 装载 T43 的状态，作为当前逻辑判断起点。
LD     T43
// 条件成立时将字数据 +3 写入 VW602。
MOVW   +3, VW602
// 装载 M10.5 的状态，作为当前逻辑判断起点。
LD     M10.5
// 与 T62 进行串联条件判断。
A      T62
// 与 M15.2 的反状态进行串联条件判断。
AN     M15.2
// 条件成立时置位 M15.2，连续置位 1 位。
S      M15.2, 1
// 条件成立时置位 M10.6，连续置位 1 位。
S      M10.6, 1
// 条件成立时置位 M29.0，连续置位 1 位。
S      M29.0, 1
Network 92
// 程序网络 92：满足条件时执行批量复位/停止处理。
// 装载 M12.5 的状态，作为当前逻辑判断起点。
LD     M12.5
// 条件成立时复位 M10.5，连续复位 1 位。
R      M10.5, 1
// 条件成立时复位 M29.2，连续复位 1 位。
R      M29.2, 1
Network 93
// 程序网络 93：执行流程条件判断与状态控制。
// 装载 M12.5 的状态，作为当前逻辑判断起点。
LD     M12.5
// 条件成立时置位 M15.3，连续置位 1 位。
S      M15.3, 1
Network 94
// 程序网络 94：执行流程条件判断与状态控制。
// 装载 T51 的状态，作为当前逻辑判断起点。
LD     T51
// 条件成立时复位 M14.3，连续复位 1 位。
R      M14.3, 1
Network 95
// 程序网络 95：执行流程条件判断与状态控制。
// 装载 T51 的状态，作为当前逻辑判断起点。
LD     T51
// 条件成立时复位 Q0.6，连续复位 1 位。
R      Q0.6, 1
Network 96
// 程序网络 96：满足条件时置位多个流程状态。
// 装载 M12.5 的状态，作为当前逻辑判断起点。
LD     M12.5
// 条件成立时置位 M21.5，连续置位 1 位。
S      M21.5, 1
// 条件成立时置位 M22.7，连续置位 1 位。
S      M22.7, 1
Network 97
// 程序网络 97：更新流程状态字或显示/通讯状态值。
// 装载 M12.5 的状态，作为当前逻辑判断起点。
LD     M12.5
// 条件成立时将字数据 +3 写入 VW600。
MOVW   +3, VW600
Network 98
// 程序网络 98：更新流程状态字或显示/通讯状态值。
// 装载 M12.5 的状态，作为当前逻辑判断起点。
LD     M12.5
// 条件成立时将字数据 +3 写入 VW602。
MOVW   +3, VW602
Network 99
// 程序网络 99：满足条件时执行批量复位/停止处理。
// 装载 M12.6 的状态，作为当前逻辑判断起点。
LD     M12.6
// 条件成立时复位 M10.6，连续复位 1 位。
R      M10.6, 1
// 条件成立时复位 M29.0，连续复位 1 位。
R      M29.0, 1
// 条件成立时置位 Q0.6，连续置位 1 位。
S      Q0.6, 1
Network 100
// 程序网络 100：执行流程条件判断与状态控制。
// 装载 M12.6 的状态，作为当前逻辑判断起点。
LD     M12.6
// 条件成立时置位 M14.4，连续置位 1 位。
S      M14.4, 1
Network 101
// 程序网络 101：满足条件时执行批量复位/停止处理。
// 装载 T52 的状态，作为当前逻辑判断起点。
LD     T52
// 条件成立时复位 M14.4，连续复位 1 位。
R      M14.4, 1
// 条件成立时复位 M15.2，连续复位 2 位。
R      M15.2, 2
Network 102
// 程序网络 102：满足条件时置位多个流程状态。
// 装载 T52 的状态，作为当前逻辑判断起点。
LD     T52
// 条件成立时置位 M10.7，连续置位 1 位。
S      M10.7, 1
// 条件成立时置位 M29.1，连续置位 1 位。
S      M29.1, 1
Network 103
// 程序网络 103：执行流程条件判断与状态控制。
// 装载 M12.6 的状态，作为当前逻辑判断起点。
LD     M12.6
// 条件成立时置位 M22.7，连续置位 1 位。
S      M22.7, 1
Network 104
// 程序网络 104：更新流程状态字或显示/通讯状态值。
// 装载 M12.6 的状态，作为当前逻辑判断起点。
LD     M12.6
// 条件成立时将字数据 +3 写入 VW602。
MOVW   +3, VW602
Network 105
// 程序网络 105：执行流程条件判断与状态控制。
// 装载 M12.7 的状态，作为当前逻辑判断起点。
LD     M12.7
// 条件成立时复位 M10.7，连续复位 1 位。
R      M10.7, 1
Network 106
// 程序网络 106：执行流程条件判断与状态控制。
// 装载 M12.7 的状态，作为当前逻辑判断起点。
LD     M12.7
R      M29.1, 1
// 条件成立时置位 M15.1，连续置位 1 位。
S      M15.1, 1
Network 107
// 程序网络 107：执行流程条件判断与状态控制。
// 装载 M12.7 的状态，作为当前逻辑判断起点。
LD     M12.7
// 条件成立时置位 M22.6，连续置位 1 位。
S      M22.6, 1
Network 108
// 程序网络 108：爆闪位夹具稳定等待结束后，进入五次爆闪工序 M11.0。
// 夹紧下压完成后等待 T38 到时，再启动 Flash 测试。
// 装载 M12.7 的状态，作为当前逻辑判断起点。
LD     M12.7
// 条件成立时将字数据 +3 写入 VW602。
MOVW   +3, VW602
// 装载 T38 的状态，作为当前逻辑判断起点。
LD     T38
// 与 M15.1 进行串联条件判断。
A      M15.1
// 条件成立时复位 M15.1，连续复位 1 位。
R      M15.1, 1
// 条件成立时置位 M11.0，连续置位 1 位。
S      M11.0, 1
// ----------------------------------------------------------------------
// 五次爆闪测试：双爆闪灯按五个发光脉冲同步动作
// ----------------------------------------------------------------------
Network 109
// 程序网络 109：满足条件时执行批量复位/停止处理。
// 装载 M11.0 的反状态，作为当前逻辑判断起点。
LDN    M11.0
// 条件成立时复位 M13.5，连续复位 3 位。
R      M13.5, 3
// 条件成立时复位 M14.5，连续复位 3 位。
R      M14.5, 3
// 条件成立时复位 M15.4，连续复位 4 位。
R      M15.4, 4
Network 110
// 程序网络 110：五次爆闪工序开始时启动第1个发光子步 M13.5。
// 装载 M11.0 的状态，作为当前逻辑判断起点。
LD     M11.0
// 与 M13.5 的反状态进行串联条件判断。
AN     M13.5
// 与 M13.6 的反状态进行串联条件判断。
AN     M13.6
// 与 M13.7 的反状态进行串联条件判断。
AN     M13.7
// 与 M14.5 的反状态进行串联条件判断。
AN     M14.5
// 与 M14.6 的反状态进行串联条件判断。
AN     M14.6
// 与 M14.7 的反状态进行串联条件判断。
AN     M14.7
// 与 M15.4 的反状态进行串联条件判断。
AN     M15.4
// 与 M15.5 的反状态进行串联条件判断。
AN     M15.5
// 与 M15.6 的反状态进行串联条件判断。
AN     M15.6
// 与 M15.7 的反状态进行串联条件判断。
AN     M15.7
// 条件成立时置位 M13.5，连续置位 1 位。
S      M13.5, 1
Network 111
// 程序网络 111：定时与条件控制，涉及 T53。
// 装载 M13.5 的状态，作为当前逻辑判断起点。
LD     M13.5
// T53（五次爆闪第1个亮灯段）：PT=+10，时间基准=100 ms，实际延迟=1.0秒。
TON    T53, +10
Network 112
// 程序网络 112：执行流程条件判断与状态控制。
// 装载 T53 的状态，作为当前逻辑判断起点。
LD     T53
// 条件成立时复位 M13.5，连续复位 1 位。
R      M13.5, 1
Network 113
// 程序网络 113：执行流程条件判断与状态控制。
// 装载 T53 的状态，作为当前逻辑判断起点。
LD     T53
// 条件成立时置位 M13.6，连续置位 1 位。
S      M13.6, 1
Network 114
// 程序网络 114：定时与条件控制，涉及 T54。
// 装载 M13.6 的状态，作为当前逻辑判断起点。
LD     M13.6
// T54（第1次与第2次爆闪间隔）：PT=+10，时间基准=100 ms，实际延迟=1.0秒。
TON    T54, +10
Network 115
// 程序网络 115：执行流程条件判断与状态控制。
// 装载 T54 的状态，作为当前逻辑判断起点。
LD     T54
// 条件成立时复位 M13.6，连续复位 1 位。
R      M13.6, 1
Network 116
// 程序网络 116：执行流程条件判断与状态控制。
// 装载 T54 的状态，作为当前逻辑判断起点。
LD     T54
// 条件成立时置位 M13.7，连续置位 1 位。
S      M13.7, 1
Network 117
// 程序网络 117：定时与条件控制，涉及 T55。
// 装载 M13.7 的状态，作为当前逻辑判断起点。
LD     M13.7
// T55（五次爆闪第2个亮灯段）：PT=+10，时间基准=100 ms，实际延迟=1.0秒。
TON    T55, +10
Network 118
// 程序网络 118：执行流程条件判断与状态控制。
// 装载 T55 的状态，作为当前逻辑判断起点。
LD     T55
// 条件成立时复位 M13.7，连续复位 1 位。
R      M13.7, 1
Network 119
// 程序网络 119：执行流程条件判断与状态控制。
// 装载 T55 的状态，作为当前逻辑判断起点。
LD     T55
// 条件成立时置位 M14.5，连续置位 1 位。
S      M14.5, 1
Network 120
// 程序网络 120：定时与条件控制，涉及 T56。
// 装载 M14.5 的状态，作为当前逻辑判断起点。
LD     M14.5
// T56（第2次与第3次爆闪间隔）：PT=+10，时间基准=100 ms，实际延迟=1.0秒。
TON    T56, +10
Network 121
// 程序网络 121：执行流程条件判断与状态控制。
// 装载 T56 的状态，作为当前逻辑判断起点。
LD     T56
// 条件成立时复位 M14.5，连续复位 1 位。
R      M14.5, 1
Network 122
// 程序网络 122：执行流程条件判断与状态控制。
// 装载 T56 的状态，作为当前逻辑判断起点。
LD     T56
// 条件成立时置位 M14.6，连续置位 1 位。
S      M14.6, 1
Network 123
// 程序网络 123：定时与条件控制，涉及 T57。
// 装载 M14.6 的状态，作为当前逻辑判断起点。
LD     M14.6
// T57（五次爆闪第3个亮灯段）：PT=+10，时间基准=100 ms，实际延迟=1.0秒。
TON    T57, +10
Network 124
// 程序网络 124：执行流程条件判断与状态控制。
// 装载 T57 的状态，作为当前逻辑判断起点。
LD     T57
// 条件成立时复位 M14.6，连续复位 1 位。
R      M14.6, 1
Network 125
// 程序网络 125：执行流程条件判断与状态控制。
// 装载 T57 的状态，作为当前逻辑判断起点。
LD     T57
// 条件成立时置位 M14.7，连续置位 1 位。
S      M14.7, 1
Network 126
// 程序网络 126：定时与条件控制，涉及 T58。
// 装载 M14.7 的状态，作为当前逻辑判断起点。
LD     M14.7
// T58（第3次与第4次爆闪间隔）：PT=+10，时间基准=100 ms，实际延迟=1.0秒。
TON    T58, +10
Network 127
// 程序网络 127：执行流程条件判断与状态控制。
// 装载 T58 的状态，作为当前逻辑判断起点。
LD     T58
// 条件成立时复位 M14.7，连续复位 1 位。
R      M14.7, 1
Network 128
// 程序网络 128：执行流程条件判断与状态控制。
// 装载 T58 的状态，作为当前逻辑判断起点。
LD     T58
// 条件成立时置位 M15.4，连续置位 1 位。
S      M15.4, 1
Network 129
// 程序网络 129：定时与条件控制，涉及 T59。
// 装载 M15.4 的状态，作为当前逻辑判断起点。
LD     M15.4
// T59（五次爆闪第4个亮灯段）：PT=+10，时间基准=100 ms，实际延迟=1.0秒。
TON    T59, +10
Network 130
// 程序网络 130：执行流程条件判断与状态控制。
// 装载 T59 的状态，作为当前逻辑判断起点。
LD     T59
// 条件成立时复位 M15.4，连续复位 1 位。
R      M15.4, 1
Network 131
// 程序网络 131：执行流程条件判断与状态控制。
// 装载 T59 的状态，作为当前逻辑判断起点。
LD     T59
// 条件成立时置位 M15.5，连续置位 1 位。
S      M15.5, 1
Network 132
// 程序网络 132：定时与条件控制，涉及 T60。
// 装载 M15.5 的状态，作为当前逻辑判断起点。
LD     M15.5
// T60（第4次与第5次爆闪间隔）：PT=+10，时间基准=100 ms，实际延迟=1.0秒。
TON    T60, +10
Network 133
// 程序网络 133：执行流程条件判断与状态控制。
// 装载 T60 的状态，作为当前逻辑判断起点。
LD     T60
// 条件成立时复位 M15.5，连续复位 1 位。
R      M15.5, 1
Network 134
// 程序网络 134：执行流程条件判断与状态控制。
// 装载 T60 的状态，作为当前逻辑判断起点。
LD     T60
// 条件成立时置位 M15.6，连续置位 1 位。
S      M15.6, 1
Network 135
// 程序网络 135：定时与条件控制，涉及 T61。
// 装载 M15.6 的状态，作为当前逻辑判断起点。
LD     M15.6
// T61（五次爆闪第5个亮灯段）：PT=+10，时间基准=100 ms，实际延迟=1.0秒。
TON    T61, +10
Network 136
// 程序网络 136：执行流程条件判断与状态控制。
// 装载 T61 的状态，作为当前逻辑判断起点。
LD     T61
// 条件成立时复位 M15.6，连续复位 1 位。
R      M15.6, 1
Network 137
// 程序网络 137：执行流程条件判断与状态控制。
// 装载 T61 的状态，作为当前逻辑判断起点。
LD     T61
// 条件成立时置位 M15.7，连续置位 1 位。
S      M15.7, 1
// ----------------------------------------------------------------------
// 爆闪结束 -> 电磁干扰 -> 回初始位
// ----------------------------------------------------------------------
Network 138
// 程序网络 138：第5次爆闪结束，关闭爆闪输出并转入电磁干扰工序 M11.2。
// 装载 M15.7 的状态，作为当前逻辑判断起点。
LD     M15.7
// 条件成立时复位 M15.7，连续复位 1 位。
R      M15.7, 1
// 条件成立时复位 M11.0，连续复位 1 位。
R      M11.0, 1
// 条件成立时置位 M11.2，连续置位 1 位。
S      M11.2, 1
// 条件成立时复位 M29.0，连续复位 8 位。
R      M29.0, 8
// 条件成立时复位 M30.5，连续复位 1 位。
R      M30.5, 1
// 条件成立时复位 M30.6，连续复位 1 位。
R      M30.6, 1
// 条件成立时复位 Q1.2，连续复位 1 位。
R      Q1.2, 1
// 条件成立时复位 Q1.3，连续复位 1 位。
R      Q1.3, 1
// 条件成立时置位 M23.0，连续置位 1 位。
S      M23.0, 1
// 条件成立时置位 M21.6，连续置位 1 位。
S      M21.6, 1
// 条件成立时将字数据 +4 写入 VW600。
MOVW   +4, VW600
// 条件成立时将字数据 +3 写入 VW602。
MOVW   +3, VW602
Network 139
// 程序网络 139：执行流程条件判断与状态控制。
// 装载 M11.1 的状态，作为当前逻辑判断起点。
LD     M11.1
// 条件成立时置位 M11.2，连续置位 1 位。
S      M11.2, 1
Network 140
// 程序网络 140：执行流程条件判断与状态控制。
// 装载 M11.1 的状态，作为当前逻辑判断起点。
LD     M11.1
// 条件成立时复位 M11.1，连续复位 1 位。
R      M11.1, 1
Network 141
// 程序网络 141：执行流程条件判断与状态控制。
// 装载 M11.2 的状态，作为当前逻辑判断起点。
LD     M11.2
// 条件成立时置位 M23.1，连续置位 1 位。
S      M23.1, 1
Network 142
// 程序网络 142：电磁干扰继电器保持计时 T39；期间 M11.2 经安全门驱动 Q0.7。
// 装载 M11.2 的状态，作为当前逻辑判断起点。
LD     M11.2
// T39（电磁干扰继电器保持时间）：PT=+100，时间基准=100 ms，实际延迟=10.0秒。
TON    T39, +100
Network 143
// 程序网络 143：执行流程条件判断与状态控制。
// 装载 T39 的状态，作为当前逻辑判断起点。
LD     T39
// 条件成立时复位 M11.2，连续复位 1 位。
R      M11.2, 1
Network 144
// 程序网络 144：电磁干扰结束，清动作并进入回初始位流程 M11.4/M10.0。
// 装载 T39 的状态，作为当前逻辑判断起点。
LD     T39
// 条件成立时复位 M10.0，连续复位 12 位。
R      M10.0, 12
// 条件成立时复位 M13.0，连续复位 8 位。
R      M13.0, 8
// 条件成立时复位 M14.0，连续复位 8 位。
R      M14.0, 8
// 条件成立时复位 M15.0，连续复位 4 位。
R      M15.0, 4
// 条件成立时复位 M29.0，连续复位 8 位。
R      M29.0, 8
// 条件成立时复位 M30.0，连续复位 8 位。
R      M30.0, 8
// 条件成立时复位 Q0.0，连续复位 8 位。
R      Q0.0, 8
// 条件成立时复位 Q1.0，连续复位 4 位。
R      Q1.0, 4
// 条件成立时置位 M11.4，连续置位 1 位。
S      M11.4, 1
// 条件成立时置位 M10.0，连续置位 1 位。
S      M10.0, 1
// 条件成立时置位 M29.2，连续置位 1 位。
S      M29.2, 1
Network 145
// 程序网络 145：执行流程条件判断与状态控制。
// 装载 T39 的状态，作为当前逻辑判断起点。
LD     T39
// 条件成立时置位 M23.2，连续置位 1 位。
S      M23.2, 1
Network 146
// 程序网络 146：执行流程条件判断与状态控制。
// 装载 T39 的状态，作为当前逻辑判断起点。
LD     T39
// 条件成立时置位 M23.3，连续置位 1 位。
S      M23.3, 1
Network 147
// 程序网络 147：执行流程条件判断与状态控制。
// 装载 T39 的状态，作为当前逻辑判断起点。
LD     T39
// 条件成立时置位 M21.7，连续置位 1 位。
S      M21.7, 1
Network 148
// 程序网络 148：更新流程状态字或显示/通讯状态值。
// 装载 T39 的状态，作为当前逻辑判断起点。
LD     T39
// 条件成立时将字数据 +1 写入 VW600。
MOVW   +1, VW600
// 条件成立时将字数据 +1 写入 VW602。
MOVW   +1, VW602
// ----------------------------------------------------------------------
// 回零完成、自动流程结束及完成状态锁存
// ----------------------------------------------------------------------
Network 149
// 程序网络 149：回初始位完成后锁存流程完成 M0.1，并清除动作及输出命令。
// 装载 M11.3 的状态，作为当前逻辑判断起点。
LD     M11.3
// 条件成立时置位 M0.1，连续置位 1 位。
S      M0.1, 1
// 条件成立时复位 M21.0，连续复位 8 位。
R      M21.0, 8
// 条件成立时复位 M22.0，连续复位 12 位。
R      M22.0, 12
// 条件成立时复位 M29.0，连续复位 8 位。
R      M29.0, 8
// 条件成立时复位 M30.0，连续复位 8 位。
R      M30.0, 8
// 条件成立时复位 Q0.0，连续复位 8 位。
R      Q0.0, 8
// 条件成立时复位 Q1.0，连续复位 4 位。
R      Q1.0, 4
Network 150
// 程序网络 150：执行流程条件判断与状态控制。
// 装载 M11.3 的状态，作为当前逻辑判断起点。
LD     M11.3
// 条件成立时复位 M0.0，连续复位 1 位。
R      M0.0, 1
Network 151
// 程序网络 151：执行流程条件判断与状态控制。
// 装载 M11.3 的状态，作为当前逻辑判断起点。
LD     M11.3
// 条件成立时复位 M11.3，连续复位 1 位。
R      M11.3, 1
Network 152
// 程序网络 152：更新流程状态字或显示/通讯状态值。
// 装载 M0.1 的状态，作为当前逻辑判断起点。
LD     M0.1
// 条件成立时将字数据 +0 写入 VW600。
MOVW   +0, VW600
Network 153
// 程序网络 153：更新流程状态字或显示/通讯状态值。
// 装载 M0.1 的状态，作为当前逻辑判断起点。
LD     M0.1
// 条件成立时将字数据 +0 写入 VW602。
MOVW   +0, VW602
// ----------------------------------------------------------------------
// VW600/VW602 上位机工序阶段码维护
// ----------------------------------------------------------------------
Network 154
// 程序网络 154：更新流程状态字或显示/通讯状态值。
// 装载 M10.0 的状态，作为当前逻辑判断起点。
LD     M10.0
// 条件成立时将字数据 +1 写入 VW600。
MOVW   +1, VW600
// 条件成立时将字数据 +1 写入 VW602。
MOVW   +1, VW602
Network 155
// 程序网络 155：更新流程状态字或显示/通讯状态值。
// 装载 M14.0 的状态，作为当前逻辑判断起点。
LD     M14.0
// 与 M10.1 进行并联“或”条件判断。
O      M10.1
// 条件成立时将字数据 +1 写入 VW600。
MOVW   +1, VW600
// 条件成立时将字数据 +1 写入 VW602。
MOVW   +1, VW602
Network 156
// 程序网络 156：更新流程状态字或显示/通讯状态值。
// 装载 M14.1 的状态，作为当前逻辑判断起点。
LD     M14.1
// 与 M10.2 进行并联“或”条件判断。
O      M10.2
// 条件成立时将字数据 +2 写入 VW600。
MOVW   +2, VW600
// 条件成立时将字数据 +2 写入 VW602。
MOVW   +2, VW602
Network 157
// 程序网络 157：更新流程状态字或显示/通讯状态值。
// 装载 M14.2 的状态，作为当前逻辑判断起点。
LD     M14.2
// 与 M10.3 进行并联“或”条件判断。
O      M10.3
// 与 M15.0 进行并联“或”条件判断。
O      M15.0
// 条件成立时将字数据 +2 写入 VW600。
MOVW   +2, VW600
// 条件成立时将字数据 +2 写入 VW602。
MOVW   +2, VW602
Network 158
// 程序网络 158：更新流程状态字或显示/通讯状态值。
// 装载 M10.4 的状态，作为当前逻辑判断起点。
LD     M10.4
// 与 M13.0 进行并联“或”条件判断。
O      M13.0
// 与 M13.1 进行并联“或”条件判断。
O      M13.1
// 与 M13.2 进行并联“或”条件判断。
O      M13.2
// 与 M13.3 进行并联“或”条件判断。
O      M13.3
// 与 M13.4 进行并联“或”条件判断。
O      M13.4
// 条件成立时将字数据 +2 写入 VW600。
MOVW   +2, VW600
// 条件成立时将字数据 +2 写入 VW602。
MOVW   +2, VW602
Network 159
// 程序网络 159：更新流程状态字或显示/通讯状态值。
// 装载 M10.5 的状态，作为当前逻辑判断起点。
LD     M10.5
// 条件成立时将字数据 +2 写入 VW600。
MOVW   +2, VW600
// 条件成立时将字数据 +3 写入 VW602。
MOVW   +3, VW602
Network 160
// 程序网络 160：更新流程状态字或显示/通讯状态值。
// 装载 M15.2 的状态，作为当前逻辑判断起点。
LD     M15.2
// 与 M15.3 进行并联“或”条件判断。
O      M15.3
// 与 M10.6 进行并联“或”条件判断。
O      M10.6
// 条件成立时将字数据 +3 写入 VW600。
MOVW   +3, VW600
// 条件成立时将字数据 +3 写入 VW602。
MOVW   +3, VW602
Network 161
// 程序网络 161：更新流程状态字或显示/通讯状态值。
// 装载 M14.4 的状态，作为当前逻辑判断起点。
LD     M14.4
// 与 M10.7 进行并联“或”条件判断。
O      M10.7
// 条件成立时将字数据 +3 写入 VW600。
MOVW   +3, VW600
// 条件成立时将字数据 +3 写入 VW602。
MOVW   +3, VW602
Network 162
// 程序网络 162：更新流程状态字或显示/通讯状态值。
// 装载 M11.0 的状态，作为当前逻辑判断起点。
LD     M11.0
// 与 M15.1 进行并联“或”条件判断。
O      M15.1
// 条件成立时将字数据 +3 写入 VW600。
MOVW   +3, VW600
// 条件成立时将字数据 +3 写入 VW602。
MOVW   +3, VW602
Network 163
// 程序网络 163：更新流程状态字或显示/通讯状态值。
// 装载 M11.2 的状态，作为当前逻辑判断起点。
LD     M11.2
// 条件成立时将字数据 +4 写入 VW600。
MOVW   +4, VW600
// 条件成立时将字数据 +3 写入 VW602。
MOVW   +3, VW602
// ----------------------------------------------------------------------
// 上位机工序阶段汇总继电器 M21.0~M21.3
// ----------------------------------------------------------------------
Network 164
// 程序网络 164：组合条件并生成状态或输出结果。
// 装载 M10.0 的状态，作为当前逻辑判断起点。
LD     M10.0
// 与 M14.0 进行并联“或”条件判断。
O      M14.0
// 与 M10.1 进行并联“或”条件判断。
O      M10.1
// 与 M14.1 进行并联“或”条件判断。
O      M14.1
// 将当前逻辑结果写入 M21.0。
=      M21.0
Network 165
// 程序网络 165：组合条件并生成状态或输出结果。
// 装载 M10.2 的状态，作为当前逻辑判断起点。
LD     M10.2
// 与 M14.2 进行并联“或”条件判断。
O      M14.2
// 与 M10.3 进行并联“或”条件判断。
O      M10.3
// 与 M15.0 进行并联“或”条件判断。
O      M15.0
// 与 M10.4 进行并联“或”条件判断。
O      M10.4
// 与 M10.5 进行并联“或”条件判断。
O      M10.5
// 与 M14.3 进行并联“或”条件判断。
O      M14.3
// 将当前逻辑结果写入 M21.1。
=      M21.1
Network 166
// 程序网络 166：组合条件并生成状态或输出结果。
// 装载 M10.6 的状态，作为当前逻辑判断起点。
LD     M10.6
// 与 M14.4 进行并联“或”条件判断。
O      M14.4
// 与 M10.7 进行并联“或”条件判断。
O      M10.7
// 与 M11.0 进行并联“或”条件判断。
O      M11.0
// 与 M15.1 进行并联“或”条件判断。
O      M15.1
// 与 M15.2 进行并联“或”条件判断。
O      M15.2
// 与 M15.3 进行并联“或”条件判断。
O      M15.3
// 将当前逻辑结果写入 M21.2。
=      M21.2
Network 167
// 程序网络 167：组合条件并生成状态或输出结果。
// 装载 M11.2 的状态，作为当前逻辑判断起点。
LD     M11.2
// 将当前逻辑结果写入 M21.3。
=      M21.3
// ----------------------------------------------------------------------
// 自动动作 M29.0~M29.4 的下降沿检测
// ----------------------------------------------------------------------
Network 168
// 程序网络 168：组合条件并生成状态或输出结果。
// 装载 M28.0 的状态，作为当前逻辑判断起点。
LD     M28.0
// 与 M29.0 的反状态进行串联条件判断。
AN     M29.0
// 将当前逻辑结果写入 M27.0。
=      M27.0
Network 169
// 程序网络 169：组合条件并生成状态或输出结果。
// 装载 M28.1 的状态，作为当前逻辑判断起点。
LD     M28.1
// 与 M29.1 的反状态进行串联条件判断。
AN     M29.1
// 将当前逻辑结果写入 M27.1。
=      M27.1
Network 170
// 程序网络 170：组合条件并生成状态或输出结果。
// 装载 M28.2 的状态，作为当前逻辑判断起点。
LD     M28.2
// 与 M29.2 的反状态进行串联条件判断。
AN     M29.2
// 将当前逻辑结果写入 M27.2。
=      M27.2
Network 171
// 程序网络 171：组合条件并生成状态或输出结果。
// 装载 M28.3 的状态，作为当前逻辑判断起点。
LD     M28.3
// 与 M29.3 的反状态进行串联条件判断。
AN     M29.3
// 将当前逻辑结果写入 M27.3。
=      M27.3
Network 172
// 程序网络 172：组合条件并生成状态或输出结果。
// 装载 M28.4 的状态，作为当前逻辑判断起点。
LD     M28.4
// 与 M29.4 的反状态进行串联条件判断。
AN     M29.4
// 将当前逻辑结果写入 M27.4。
=      M27.4
Network 173
// 程序网络 173：组合条件并生成状态或输出结果。
// 装载 M27.1 的状态，作为当前逻辑判断起点。
LD     M27.1
// 与 M27.2 进行并联“或”条件判断。
O      M27.2
// 与 M29.1 的反状态进行串联条件判断。
AN     M29.1
// 与 M29.2 的反状态进行串联条件判断。
AN     M29.2
// 将当前逻辑结果写入 M27.5。
=      M27.5
// ----------------------------------------------------------------------
// 自动动作 M29.0~M29.4 的上升沿检测
// ----------------------------------------------------------------------
Network 174
// 程序网络 174：组合条件并生成状态或输出结果。
// 装载 M29.0 的状态，作为当前逻辑判断起点。
LD     M29.0
// 与 M28.0 的反状态进行串联条件判断。
AN     M28.0
// 将当前逻辑结果写入 M26.0。
=      M26.0
Network 175
// 程序网络 175：组合条件并生成状态或输出结果。
// 装载 M29.1 的状态，作为当前逻辑判断起点。
LD     M29.1
// 与 M28.1 的反状态进行串联条件判断。
AN     M28.1
// 将当前逻辑结果写入 M26.1。
=      M26.1
Network 176
// 程序网络 176：组合条件并生成状态或输出结果。
// 装载 M29.2 的状态，作为当前逻辑判断起点。
LD     M29.2
// 与 M28.2 的反状态进行串联条件判断。
AN     M28.2
// 将当前逻辑结果写入 M26.2。
=      M26.2
Network 177
// 程序网络 177：组合条件并生成状态或输出结果。
// 装载 M29.3 的状态，作为当前逻辑判断起点。
LD     M29.3
// 与 M28.3 的反状态进行串联条件判断。
AN     M28.3
// 将当前逻辑结果写入 M26.3。
=      M26.3
Network 178
// 程序网络 178：组合条件并生成状态或输出结果。
// 装载 M29.4 的状态，作为当前逻辑判断起点。
LD     M29.4
// 与 M28.4 的反状态进行串联条件判断。
AN     M28.4
// 将当前逻辑结果写入 M26.4。
=      M26.4
// ----------------------------------------------------------------------
// 自动动作互锁：新动作开始时撤销不兼容的旧动作
// ----------------------------------------------------------------------
Network 179
// 程序网络 179：执行流程条件判断与状态控制。
// 装载 M26.0 的状态，作为当前逻辑判断起点。
LD     M26.0
// 条件成立时复位 M29.1，连续复位 1 位。
R      M29.1, 1
Network 180
// 程序网络 180：执行流程条件判断与状态控制。
// 装载 M26.0 的状态，作为当前逻辑判断起点。
LD     M26.0
// 与 T62 的反状态进行串联条件判断。
AN     T62
// 条件成立时复位 M29.2，连续复位 1 位。
R      M29.2, 1
Network 181
// 程序网络 181：执行流程条件判断与状态控制。
// 装载 M26.0 的状态，作为当前逻辑判断起点。
LD     M26.0
// 条件成立时复位 M29.3，连续复位 1 位。
R      M29.3, 1
Network 182
// 程序网络 182：执行流程条件判断与状态控制。
// 装载 M26.0 的状态，作为当前逻辑判断起点。
LD     M26.0
// 条件成立时复位 M29.4，连续复位 1 位。
R      M29.4, 1
Network 183
// 程序网络 183：执行流程条件判断与状态控制。
// 装载 M26.1 的状态，作为当前逻辑判断起点。
LD     M26.1
// 条件成立时复位 M29.0，连续复位 1 位。
R      M29.0, 1
Network 184
// 程序网络 184：执行流程条件判断与状态控制。
// 装载 M26.1 的状态，作为当前逻辑判断起点。
LD     M26.1
// 条件成立时复位 M29.2，连续复位 1 位。
R      M29.2, 1
Network 185
// 程序网络 185：执行流程条件判断与状态控制。
// 装载 M26.1 的状态，作为当前逻辑判断起点。
LD     M26.1
// 条件成立时复位 M29.3，连续复位 1 位。
R      M29.3, 1
Network 186
// 程序网络 186：执行流程条件判断与状态控制。
// 装载 M26.1 的状态，作为当前逻辑判断起点。
LD     M26.1
// 条件成立时复位 M29.4，连续复位 1 位。
R      M29.4, 1
Network 187
// 程序网络 187：执行流程条件判断与状态控制。
// 装载 M26.2 的状态，作为当前逻辑判断起点。
LD     M26.2
// 条件成立时复位 M29.0，连续复位 1 位。
R      M29.0, 1
Network 188
// 程序网络 188：执行流程条件判断与状态控制。
// 装载 M26.2 的状态，作为当前逻辑判断起点。
LD     M26.2
// 条件成立时复位 M29.1，连续复位 1 位。
R      M29.1, 1
Network 189
// 程序网络 189：执行流程条件判断与状态控制。
// 装载 M26.2 的状态，作为当前逻辑判断起点。
LD     M26.2
// 条件成立时复位 M29.3，连续复位 1 位。
R      M29.3, 1
Network 190
// 程序网络 190：执行流程条件判断与状态控制。
// 装载 M26.2 的状态，作为当前逻辑判断起点。
LD     M26.2
// 条件成立时复位 M29.4，连续复位 1 位。
R      M29.4, 1
Network 191
// 程序网络 191：执行流程条件判断与状态控制。
// 装载 M26.3 的状态，作为当前逻辑判断起点。
LD     M26.3
// 条件成立时复位 M29.0，连续复位 1 位。
R      M29.0, 1
Network 192
// 程序网络 192：执行流程条件判断与状态控制。
// 装载 M26.3 的状态，作为当前逻辑判断起点。
LD     M26.3
// 条件成立时复位 M29.1，连续复位 1 位。
R      M29.1, 1
Network 193
// 程序网络 193：执行流程条件判断与状态控制。
// 装载 M26.3 的状态，作为当前逻辑判断起点。
LD     M26.3
// 条件成立时复位 M29.2，连续复位 1 位。
R      M29.2, 1
Network 194
// 程序网络 194：执行流程条件判断与状态控制。
// 装载 M26.3 的状态，作为当前逻辑判断起点。
LD     M26.3
// 条件成立时复位 M29.4，连续复位 1 位。
R      M29.4, 1
Network 195
// 程序网络 195：执行流程条件判断与状态控制。
// 装载 M26.4 的状态，作为当前逻辑判断起点。
LD     M26.4
// 条件成立时复位 M29.0，连续复位 1 位。
R      M29.0, 1
Network 196
// 程序网络 196：执行流程条件判断与状态控制。
// 装载 M26.4 的状态，作为当前逻辑判断起点。
LD     M26.4
// 条件成立时复位 M29.1，连续复位 1 位。
R      M29.1, 1
Network 197
// 程序网络 197：执行流程条件判断与状态控制。
// 装载 M26.4 的状态，作为当前逻辑判断起点。
LD     M26.4
// 条件成立时复位 M29.2，连续复位 1 位。
R      M29.2, 1
Network 198
// 程序网络 198：执行流程条件判断与状态控制。
// 装载 M26.4 的状态，作为当前逻辑判断起点。
LD     M26.4
// 条件成立时复位 M29.3，连续复位 1 位。
R      M29.3, 1
// ----------------------------------------------------------------------
// 自动动作切换时清理不兼容的物理输出
// ----------------------------------------------------------------------
Network 199
// 程序网络 199：执行流程条件判断与状态控制。
// 装载 M26.0 的状态，作为当前逻辑判断起点。
LD     M26.0
// 条件成立时复位 Q0.1，连续复位 1 位。
R      Q0.1, 1
Network 200
// 程序网络 200：执行流程条件判断与状态控制。
// 装载 M26.0 的状态，作为当前逻辑判断起点。
LD     M26.0
// 条件成立时复位 Q0.4，连续复位 1 位。
R      Q0.4, 1
Network 201
// 程序网络 201：执行流程条件判断与状态控制。
// 装载 M26.0 的状态，作为当前逻辑判断起点。
LD     M26.0
// 条件成立时复位 Q1.1，连续复位 1 位。
R      Q1.1, 1
Network 202
// 程序网络 202：执行流程条件判断与状态控制。
// 装载 M26.0 的状态，作为当前逻辑判断起点。
LD     M26.0
// 条件成立时复位 Q1.2，连续复位 1 位。
R      Q1.2, 1
Network 203
// 程序网络 203：执行流程条件判断与状态控制。
// 装载 M26.1 的状态，作为当前逻辑判断起点。
LD     M26.1
// 条件成立时复位 Q0.1，连续复位 1 位。
R      Q0.1, 1
Network 204
// 程序网络 204：执行流程条件判断与状态控制。
// 装载 M26.1 的状态，作为当前逻辑判断起点。
LD     M26.1
// 条件成立时复位 Q0.5，连续复位 1 位。
R      Q0.5, 1
Network 205
// 程序网络 205：执行流程条件判断与状态控制。
// 装载 M26.1 的状态，作为当前逻辑判断起点。
LD     M26.1
// 条件成立时复位 Q1.1，连续复位 1 位。
R      Q1.1, 1
Network 206
// 程序网络 206：执行流程条件判断与状态控制。
// 装载 M26.1 的状态，作为当前逻辑判断起点。
LD     M26.1
// 条件成立时复位 Q1.2，连续复位 1 位。
R      Q1.2, 1
Network 207
// 程序网络 207：执行流程条件判断与状态控制。
// 装载 M26.2 的状态，作为当前逻辑判断起点。
LD     M26.2
// 条件成立时复位 Q0.1，连续复位 1 位。
R      Q0.1, 1
Network 208
// 程序网络 208：执行流程条件判断与状态控制。
// 装载 M26.2 的状态，作为当前逻辑判断起点。
LD     M26.2
// 条件成立时复位 Q0.5，连续复位 1 位。
R      Q0.5, 1
Network 209
// 程序网络 209：执行流程条件判断与状态控制。
// 装载 M26.2 的状态，作为当前逻辑判断起点。
LD     M26.2
// 条件成立时复位 Q1.2，连续复位 1 位。
R      Q1.2, 1
Network 210
// 程序网络 210：执行流程条件判断与状态控制。
// 装载 M26.3 的状态，作为当前逻辑判断起点。
LD     M26.3
// 条件成立时复位 Q0.4，连续复位 1 位。
R      Q0.4, 1
Network 211
// 程序网络 211：执行流程条件判断与状态控制。
// 装载 M26.3 的状态，作为当前逻辑判断起点。
LD     M26.3
// 条件成立时复位 Q0.5，连续复位 1 位。
R      Q0.5, 1
Network 212
// 程序网络 212：执行流程条件判断与状态控制。
// 装载 M26.3 的状态，作为当前逻辑判断起点。
LD     M26.3
// 条件成立时复位 Q1.1，连续复位 1 位。
R      Q1.1, 1
Network 213
// 程序网络 213：执行流程条件判断与状态控制。
// 装载 M26.3 的状态，作为当前逻辑判断起点。
LD     M26.3
// 条件成立时复位 Q1.2，连续复位 1 位。
R      Q1.2, 1
Network 214
// 程序网络 214：执行流程条件判断与状态控制。
// 装载 M26.4 的状态，作为当前逻辑判断起点。
LD     M26.4
// 条件成立时复位 Q0.1，连续复位 1 位。
R      Q0.1, 1
Network 215
// 程序网络 215：执行流程条件判断与状态控制。
// 装载 M26.4 的状态，作为当前逻辑判断起点。
LD     M26.4
// 条件成立时复位 Q0.4，连续复位 1 位。
R      Q0.4, 1
Network 216
// 程序网络 216：执行流程条件判断与状态控制。
// 装载 M26.4 的状态，作为当前逻辑判断起点。
LD     M26.4
// 条件成立时复位 Q0.5，连续复位 1 位。
R      Q0.5, 1
Network 217
// 程序网络 217：执行流程条件判断与状态控制。
// 装载 M26.4 的状态，作为当前逻辑判断起点。
LD     M26.4
// 条件成立时复位 Q1.1，连续复位 1 位。
R      Q1.1, 1
// ----------------------------------------------------------------------
// 动作切换与手动总停止的集中输出清零
// ----------------------------------------------------------------------
Network 218
// 程序网络 218：组合条件并生成状态或输出结果。
// 装载 M26.0 的状态，作为当前逻辑判断起点。
LD     M26.0
// 与 M26.1 进行并联“或”条件判断。
O      M26.1
// 与 M26.2 进行并联“或”条件判断。
O      M26.2
// 与 M26.3 进行并联“或”条件判断。
O      M26.3
// 与 M26.4 进行并联“或”条件判断。
O      M26.4
// 将当前逻辑结果写入 M26.5。
=      M26.5
Network 219
// 程序网络 219：执行流程条件判断与状态控制。
// 装载 M26.5 的状态，作为当前逻辑判断起点。
LD     M26.5
// 条件成立时复位 M30.0，连续复位 7 位。
R      M30.0, 7
Network 220
// 程序网络 220：执行流程条件判断与状态控制。
// 装载 M26.5 的状态，作为当前逻辑判断起点。
LD     M26.5
// 条件成立时复位 Q0.0，连续复位 8 位。
R      Q0.0, 8
Network 221
// 程序网络 221：执行流程条件判断与状态控制。
// 装载 M26.5 的状态，作为当前逻辑判断起点。
LD     M26.5
// 条件成立时复位 Q1.0，连续复位 4 位。
R      Q1.0, 4
Network 222
// 程序网络 222：执行流程条件判断与状态控制。
// 装载 M30.7 的状态，作为当前逻辑判断起点。
LD     M30.7
// 条件成立时复位 M30.0，连续复位 8 位。
R      M30.0, 8
Network 223
// 程序网络 223：执行流程条件判断与状态控制。
// 装载 M30.7 的状态，作为当前逻辑判断起点。
LD     M30.7
// 条件成立时复位 M29.0，连续复位 8 位。
R      M29.0, 8
Network 224
// 程序网络 224：执行流程条件判断与状态控制。
// 装载 M30.7 的状态，作为当前逻辑判断起点。
LD     M30.7
// 条件成立时复位 Q0.0，连续复位 8 位。
R      Q0.0, 8
Network 225
// 程序网络 225：执行流程条件判断与状态控制。
// 装载 M30.7 的状态，作为当前逻辑判断起点。
LD     M30.7
// 条件成立时复位 Q1.0，连续复位 4 位。
R      Q1.0, 4
// ----------------------------------------------------------------------
// 自动/手动命令经安全链合成为 M31.0~M31.7
// ----------------------------------------------------------------------
Network 226
// 程序网络 226：安全链满足且未手动总停时，开放总输出安全使能 M31.7。
// 装载 M0.3 的状态，作为当前逻辑判断起点。
LD     M0.3
// 与 M30.7 的反状态进行串联条件判断。
AN     M30.7
// 将当前逻辑结果写入 M31.7。
=      M31.7
Network 227
// 程序网络 227：组合条件并生成状态或输出结果。
// 装载 M30.0 的状态，作为当前逻辑判断起点。
LD     M30.0
// 与 M15.0 进行并联“或”条件判断。
O      M15.0
// 与 M10.4 进行并联“或”条件判断。
O      M10.4
// 与 M31.7 进行串联条件判断。
A      M31.7
// 将当前逻辑结果写入 M31.0。
=      M31.0
Network 228
// 程序网络 228：组合条件并生成状态或输出结果。
// 装载 M30.1 的状态，作为当前逻辑判断起点。
LD     M30.1
// 与 M29.1 进行并联“或”条件判断。
O      M29.1
// 与 M29.2 进行并联“或”条件判断。
O      M29.2
// 与 Q0.4 进行并联“或”条件判断。
O      Q0.4
// 与 M27.5 的反状态进行串联条件判断。
AN     M27.5
// 与 M31.7 进行串联条件判断。
A      M31.7
AN     M15.0
AN     M15.1
// 将当前逻辑结果写入 M31.1。
=      M31.1
Network 229
// 程序网络 229：组合条件并生成状态或输出结果。
// 装载 M30.2 的状态，作为当前逻辑判断起点。
LD     M30.2
// 与 M29.2 进行并联“或”条件判断。
O      M29.2
// 与 Q1.1 进行并联“或”条件判断。
O      Q1.1
// 与 M29.1 的反状态进行串联条件判断。
AN     M29.1
// 与 M27.2 的反状态进行串联条件判断。
AN     M27.2
// 与 M31.7 进行串联条件判断。
A      M31.7
AN     M15.0
AN     M15.1
// 将当前逻辑结果写入 M31.2。
=      M31.2
Network 230
// 程序网络 230：组合条件并生成状态或输出结果。
// 装载 M30.3 的状态，作为当前逻辑判断起点。
LD     M30.3
// 与 M29.0 进行并联“或”条件判断。
O      M29.0
// 与 Q0.5 进行并联“或”条件判断。
O      Q0.5
// 与 M27.0 的反状态进行串联条件判断。
AN     M27.0
// 与 M10.4 的反状态进行串联条件判断。
AN     M10.4
// 与 M13.0 的反状态进行串联条件判断。
AN     M13.0
// 与 M13.1 的反状态进行串联条件判断。
AN     M13.1
// 与 M13.2 的反状态进行串联条件判断。
AN     M13.2
// 与 M13.3 的反状态进行串联条件判断。
AN     M13.3
// 与 M13.4 的反状态进行串联条件判断。
AN     M13.4
// 与 M29.3 的反状态进行串联条件判断。
AN     M29.3
// 与 Q0.1 的反状态进行串联条件判断。
AN     Q0.1
// 与 M31.7 进行串联条件判断。
A      M31.7
// 将当前逻辑结果写入 M31.3。
=      M31.3
Network 231
// 程序网络 231：组合条件并生成状态或输出结果。
// 装载 M30.4 的状态，作为当前逻辑判断起点。
LD     M30.4
// 与 Q0.6 进行并联“或”条件判断。
O      Q0.6
// 与 M31.7 进行串联条件判断。
A      M31.7
// 将当前逻辑结果写入 M31.4。
=      M31.4
Network 232
// 程序网络 232：组合条件并生成状态或输出结果。
// 装载 M30.5 的状态，作为当前逻辑判断起点。
LD     M30.5
// 与 M29.4 进行并联“或”条件判断。
O      M29.4
// 与 M11.0 的反状态进行串联条件判断。
AN     M11.0
// 与 M27.4 的反状态进行串联条件判断。
AN     M27.4
// 与 M31.7 进行串联条件判断。
A      M31.7
// 将当前逻辑结果写入 M31.5。
=      M31.5
Network 233
// 程序网络 233：组合条件并生成状态或输出结果。
// 装载 M30.6 的状态，作为当前逻辑判断起点。
LD     M30.6
// 与 M11.0 的反状态进行串联条件判断。
AN     M11.0
// 与 M31.7 进行串联条件判断。
A      M31.7
// 将当前逻辑结果写入 M31.6。
=      M31.6
// ----------------------------------------------------------------------
// 保存自动动作上一扫描状态，供沿检测使用
// ----------------------------------------------------------------------
Network 234
// 程序网络 234：组合条件并生成状态或输出结果。
// 装载 M29.0 的状态，作为当前逻辑判断起点。
LD     M29.0
// 将当前逻辑结果写入 M28.0。
=      M28.0
Network 235
// 程序网络 235：组合条件并生成状态或输出结果。
// 装载 M29.1 的状态，作为当前逻辑判断起点。
LD     M29.1
// 将当前逻辑结果写入 M28.1。
=      M28.1
Network 236
// 程序网络 236：组合条件并生成状态或输出结果。
// 装载 M29.2 的状态，作为当前逻辑判断起点。
LD     M29.2
// 将当前逻辑结果写入 M28.2。
=      M28.2
Network 237
// 程序网络 237：组合条件并生成状态或输出结果。
// 装载 M29.3 的状态，作为当前逻辑判断起点。
LD     M29.3
// 将当前逻辑结果写入 M28.3。
=      M28.3
Network 238
// 程序网络 238：组合条件并生成状态或输出结果。
// 装载 M29.4 的状态，作为当前逻辑判断起点。
LD     M29.4
// 将当前逻辑结果写入 M28.4。
=      M28.4
// ----------------------------------------------------------------------
// 最终物理输出 Q：电机、热源、气缸、爆闪灯、电磁干扰
// ----------------------------------------------------------------------
Network 239
// 程序网络 239：垂直电源合成 M31.1 -> 上下电机总电源 Q0.4。
// 装载 M31.1 的状态，作为当前逻辑判断起点。
LD     M31.1
// 将当前逻辑结果写入 Q0.4。
=      Q0.4
Network 240
// 程序网络 240：垂直方向合成 M31.2 -> Q1.1（1上/0下）。
// 装载 M31.2 的状态，作为当前逻辑判断起点。
LD     M31.2
// 将当前逻辑结果写入 Q1.1。
=      Q1.1
Network 241
// 程序网络 241：水平运行合成 M31.3 -> 左右电机运行 Q0.5。
// 装载 M31.3 的状态，作为当前逻辑判断起点。
LD     M31.3
// 将当前逻辑结果写入 Q0.5。
=      Q0.5
Network 242
// 程序网络 242：组合条件并生成状态或输出结果。
// AUTO_RUN 前 Q0.6 保持低电平；安全限位处理在后续网络中以单扫描脉冲实现。
// 装载 M0.0 的状态，作为当前逻辑判断起点。
LD     M0.0
// 与 M0.3 进行串联条件判断。
A      M0.3
// 与 Q0.5 的反状态进行串联条件判断。
AN     Q0.5
// 与 M31.4 进行并联“或”条件判断。
O      M31.4
// 与 M2.2 的反状态进行串联条件判断。
AN     M2.2
// 将当前逻辑结果写入 M25.1。
=      M25.1
Network 243
// 程序网络 243：热源输出合成 M31.0 -> 模拟人温度/热源 Q0.1。
// 装载 M31.0 的状态，作为当前逻辑判断起点。
LD     M31.0
// 将当前逻辑结果写入 Q0.1。
=      Q0.1
Network 244
// 程序网络 244：手动或自动挥手命令经安全门 -> 气缸/挥手测试 Q1.0。
// 装载 M30.0 的状态，作为当前逻辑判断起点。
LD     M30.0
// 与 M29.3 进行并联“或”条件判断。
O      M29.3
// 与 M31.7 进行串联条件判断。
A      M31.7
// 将当前逻辑结果写入 Q1.0。
=      Q1.0
Network 245
// 程序网络 245：手动/自动爆闪命令与五次爆闪发光子步 -> 爆闪灯1 Q1.2。
// 装载 M31.5 的状态，作为当前逻辑判断起点。
LD     M31.5
// 与 M13.5 进行并联“或”条件判断。
O      M13.5
// 与 M13.7 进行并联“或”条件判断。
O      M13.7
// 与 M14.6 进行并联“或”条件判断。
O      M14.6
// 与 M15.4 进行并联“或”条件判断。
O      M15.4
// 与 M15.6 进行并联“或”条件判断。
O      M15.6
// 与 M31.7 进行串联条件判断。
A      M31.7
// 将当前逻辑结果写入 Q1.2。
=      Q1.2
Network 246
// 程序网络 246：手动爆闪命令与五次爆闪发光子步 -> 爆闪灯2 Q1.3。
// 装载 M31.6 的状态，作为当前逻辑判断起点。
LD     M31.6
// 与 M13.5 进行并联“或”条件判断。
O      M13.5
// 与 M13.7 进行并联“或”条件判断。
O      M13.7
// 与 M14.6 进行并联“或”条件判断。
O      M14.6
// 与 M15.4 进行并联“或”条件判断。
O      M15.4
// 与 M15.6 进行并联“或”条件判断。
O      M15.6
// 与 M31.7 进行串联条件判断。
A      M31.7
// 将当前逻辑结果写入 Q1.3。
=      Q1.3
Network 247
// 程序网络 247：电磁工序位 M11.2 经输出安全使能 M31.7 -> 电磁干扰继电器 Q0.7。
// 电磁工序继电器输出控制。
// 装载 M11.2 的状态，作为当前逻辑判断起点。
LD     M11.2
// 与 M31.7 进行串联条件判断。
A      M31.7
// 将当前逻辑结果写入 Q0.7。
=      Q0.7
// ----------------------------------------------------------------------
// 安全限位处理：危险状态清输出，水平停止仅发单扫描脉冲
// ----------------------------------------------------------------------
Network 248
// 程序网络 248：执行流程条件判断与状态控制。
// 装载 M0.3 的反状态，作为当前逻辑判断起点。
LDN    M0.3
// 与 M2.2 进行串联条件判断。
A      M2.2
// 与 M2.4 的反状态进行串联条件判断。
AN     M2.4
// 条件成立时复位 Q0.0，连续复位 8 位。
R      Q0.0, 8
Network 249
// 程序网络 249：执行流程条件判断与状态控制。
// 装载 M0.3 的反状态，作为当前逻辑判断起点。
LDN    M0.3
// 与 M2.2 进行串联条件判断。
A      M2.2
// 与 M2.4 的反状态进行串联条件判断。
AN     M2.4
// 条件成立时复位 Q1.0，连续复位 4 位。
R      Q1.0, 4
Network 250
// 程序网络 250：组合条件并生成状态或输出结果。
// Q0.6 安全限位停止：检测上升沿并形成单扫描脉冲，不保持 Q0.6。
// 装载 M2.2 的状态，作为当前逻辑判断起点。
LD     M2.2
// 检测当前逻辑结果的上升沿，仅在上升沿扫描周期成立。
EU
// 将当前逻辑结果写入 M25.0。
=      M25.0
Network 251
// 程序网络 251：正常停止请求或安全限位单扫描脉冲 -> 左右电机停止 Q0.6。
// Q0.6 最终输出由正常停止请求或安全单扫描脉冲共同决定。
// 装载 M25.1 的状态，作为当前逻辑判断起点。
LD     M25.1
// 与 M25.0 进行并联“或”条件判断。
O      M25.0
// 将当前逻辑结果写入 Q0.6。
=      Q0.6
// ----------------------------------------------------------------------
// 急停兜底：清空全部工序和输出，并保持水平停止
// ----------------------------------------------------------------------
Network 252
// 程序网络 252：满足条件时执行批量复位/停止处理。
// I1.0 急停有效时，复位全部流程命令及相关物理输出。
// 装载 I1.0 的反状态，作为当前逻辑判断起点。
LDN    I1.0
// 条件成立时复位 M0.0，连续复位 1 位。
R      M0.0, 1
// 条件成立时复位 M10.0，连续复位 12 位。
R      M10.0, 12
// 条件成立时复位 M11.4，连续复位 1 位。
R      M11.4, 1
// 条件成立时复位 M12.0，连续复位 10 位。
R      M12.0, 10
// 条件成立时复位 M13.0，连续复位 8 位。
R      M13.0, 8
// 条件成立时复位 M14.0，连续复位 8 位。
R      M14.0, 8
// 条件成立时复位 M15.0，连续复位 8 位。
R      M15.0, 8
// 条件成立时复位 M21.0，连续复位 8 位。
R      M21.0, 8
// 条件成立时复位 M22.0，连续复位 12 位。
R      M22.0, 12
// 条件成立时复位 M29.0，连续复位 8 位。
R      M29.0, 8
// 条件成立时复位 M30.0，连续复位 8 位。
R      M30.0, 8
// 条件成立时复位 Q0.0，连续复位 8 位。
R      Q0.0, 8
// 条件成立时复位 Q1.0，连续复位 4 位。
R      Q1.0, 4
Network 253
// 程序网络 253：执行流程条件判断与状态控制。
// I1.0 急停期间持续置位水平停止继电器 Q0.6。
// 装载 I1.0 的反状态，作为当前逻辑判断起点。
LDN    I1.0
// 条件成立时置位 Q0.6，连续置位 1 位。
S      Q0.6, 1
// 结束主程序扫描逻辑。
END
END_ORGANIZATION_BLOCK
